{attribute 'linkalways'} 
{attribute 'no_explicit_call' := 'This FB is a CLASS and must be accessed using methods or properties'}
{attribute 'enable_dynamic_creation'}
FUNCTION_BLOCK Node_F_VN_DrawLine_TcVnVector4_DINT EXTENDS VisionNode
VAR
    aLine : _TcVnVector4_DINT;
    ipDestImage : _ITcVnImage;
    aColor : _TcVnVector4_LREAL;
    nThickness : _DINT(1);
    hrPrev : _HRESULT(S_OK);
	hresult : _HRESULT(S_OK);
END_VAR

METHOD PUBLIC  Clone : I_Node
VAR
	pNode : POINTER TO Node_F_VN_DrawLine_TcVnVector4_DINT;
END_VAR
pNode := __NEW(Node_F_VN_DrawLine_TcVnVector4_DINT);
Clone := pNode^;
END_METHOD

METHOD FB_init : BOOL
VAR_INPUT
	bInitRetains : BOOL; // if TRUE, the retain variables are initialized (warm start / cold start)
	bInCopyCode : BOOL;  // if TRUE, the instance afterwards gets moved into the copy code (online change)
END_VAR
AddInput('aLine', aLine);
AddInput('ipDestImage', ipDestImage);
AddInput('aColor', aColor);
AddInput('hrPrev', hrPrev);
AddOutput('ipDestImage', ipDestImage);
AddOutput('hresult',hresult);
AddParameter('nThickness', nThickness);
END_METHOD

METHOD PROTECTED OnExecute
hresult.Value := F_VN_DrawLine_TcVnVector4_DINT(
    aLine := aLine.Value,
	ipDestImage := ipDestImage.Value,
    aColor := aColor.Value,
    nThickness := nThickness.Value,
	hrPrev:= hrPrev.Value);
END_METHOD

METHOD PUBLIC PreExecutionCheck
VAR_INPUT
	Check : I_PreExecutionChecks;
END_VAR
Check.IsTrue(ipDestImage.IsValid, 'ipDestImage must contain an image');
Check.IsTrue(nThickness.Value >= 1, 'nThickness must be greater than or equal to 1');
END_METHOD

END_FUNCTION_BLOCK

(* stored: Version 1.1.0.1, ProductVersion 3.1.4024.15
   POU Node_F_VN_DrawLine_TcVnVector4_DINT: Id {ce120e83-5b46-04c0-21e1-d853ba4bb42b}, SpecialFunc None
   Folder Constructor: Id {fd6014e5-4fe2-0775-1e46-9045ce15263f}
   Method Clone: Id {aeafb0db-263b-0e80-0bb6-61e378333e1c}
   Method FB_init: Id {01f49f2b-3111-0b3b-1f12-fc25189f990d}
   Method OnExecute: Id {a1c03449-6b64-02b4-11d9-385017ded1e9}
   Method PreExecutionCheck: Id {453dc49b-dbb8-03f6-056a-a1a18498b476} *)
